{attribute 'qualified_only'}
VAR_GLOBAL
	tTaskCycleTime			: TIME := T#50MS;
END_VAR

(* stored: Version 1.1.0.1, ProductVersion 3.1.4024.9
   GVL GlobalVariables: Id {6788d4df-6748-4531-b252-d77ca020c340} *)
